// Mitsubishi GX Works2 project: solvvNpress_4   PLC: Q03UDV

PROGRAM MAIN
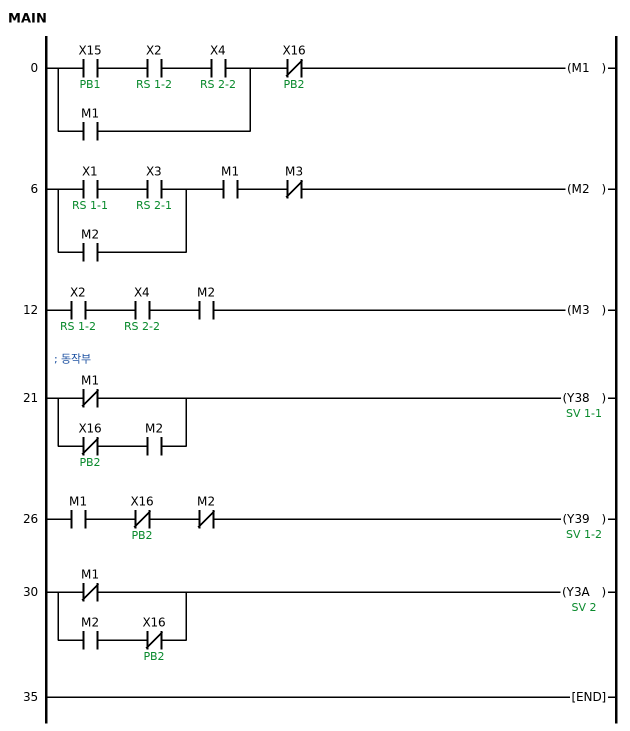
0     LD      X15  ; PB1
      AND     X2  ; RS 1-2
      AND     X4  ; RS 2-2
      OR      M1
      ANI     X16  ; PB2
      OUT     M1
6     LD      X1  ; RS 1-1
      AND     X3  ; RS 2-1
      OR      M2
      AND     M1
      ANI     M3
      OUT     M2
12    LD      X2  ; RS 1-2
      AND     X4  ; RS 2-2
      AND     M2
      OUT     M3
; 동작부
21    LDI     M1
      LDI     X16  ; PB2
      AND     M2
      ORB
      OUT     Y38  ; SV 1-1
26    LD      M1
      ANI     X16  ; PB2
      ANI     M2
      OUT     Y39  ; SV 1-2
30    LDI     M1
      LD      M2
      ANI     X16  ; PB2
      ORB
      OUT     Y3A  ; SV 2
35    END
END_PROGRAM

// device comments not shown above
X17  ; PB3
X18  ; PB4
X19  ; PB5
Y30  ; LAMP1
Y31  ; LAMP2
Y3B  ; SV 3
